PROGRAM MAIN
VAR
END_VAR

END_PROGRAM

(* stored: Version 1.1.0.1
   POU MAIN: Id {acfe357a-a3b4-4988-8542-f65080306669} *)
